KUKA KRL program: mixsort_main.src, mixsort_main.dat

--- mixsort_main.src ---
&ACCESS RVP
&REL 20
&COMMENT MixSort Main
&PARAM EDITMASK = *
&PARAM DISKPATH = KRC:\R1\Program\MixSortMain
DEF  mixsort_main ( )
;***********************************************************
;
; Copyright 2018 - 2025 speedbot All Rights reserved.
;
; File Name: mixsort_main.DAT
;
; Description:
;   Language             ==   Krl for KUKA ROBOT
;   Date                 ==   2022 - 06 - 27
;   Modification Data    ==   2025 - 02 - 10
;
; Author: speedbot
;
; Version: 1.1
;***********************************************************
;FOLD INI;%{PE}
    ;FOLD BASISTECH INI
        GLOBAL INTERRUPT DECL 3 WHEN $STOPMESS==TRUE DO IR_STOPM ( )
        INTERRUPT ON 3
        BAS (#INITMOV,0 )
    ;ENDFOLD (BASISTECH INI)
    ;FOLD USER INI
        ;Make your modifications here

    ;ENDFOLD (USER INI)
;ENDFOLD (INI)
;FOLD Basic.Override IN Override: 30  ;%{PE}
override_(30)
;ENDFOLD
;FOLD PLC.Pounce ;%{PE}
pounce_()
;ENDFOLD
mixsort_config()
;FOLD MixSort.MixSortSr ;%{PE}
mixsort_sr_inte()
;ENDFOLD
;FOLD MixSort.GetTask ;%{PE}
mixsort_get_task()
;ENDFOLD
LOOP
    continue
    wait for ToRobotFlg
    ToRobotFlg = false

    switch ToRobotAck
    case #TO_TP_NEXT
        mixsort_waitpos()
    case #TO_TP_PICT
        mixsort_picture()
    case #TO_TP_PK
        switch (GlobalTaskId)
        case 2
            mixsort_pick01()
        case 3
            mixsort_pick02()
        case 4
            mixsort_pick03()
        case 101
            mixsort_pick04()
        case 102
            mixsort_pick05()
        default
            log_error_("Unkonwn GlobalTaskId!")
        endswitch
        if (GlobalTaskId == 2) and (NOT $flag[F_PICKING]) THEN
            WAIT SEC 1
            mixsort_get_task()
        ELSE
            $flag[F_PICKING] = TRUE
            mixsort_place_select()
        ENDIF
    case #TO_TP_HOME
        exit
    endswitch
ENDLOOP
;FOLD PLC.MoveToHome ;%{PE}
move_to_home_()
;ENDFOLD
END

--- mixsort_main.dat ---
&ACCESS RVP
&REL 20
&COMMENT MixSort Main
&PARAM EDITMASK = *
&PARAM DISKPATH = KRC:\R1\Program\MixSortMain
DEFDAT  MIXSORT_MAIN
;***********************************************************
;
; Copyright 2018 - 2025 speedbot All Rights reserved.
;
; File Name: mixsort_main.DAT
;
; Description:
;   Language             ==   Krl for KUKA ROBOT
;   Date                 ==   2022 - 06 - 27
;   Modification Data    ==   2025 - 02 - 10
;
; Author: speedbot
;
; Version: 1.1
;***********************************************************
;FOLD EXTERNAL DECLARATIONS;%{PE}%MKUKATPBASIS,%CEXT,%VCOMMON,%P
;FOLD BASISTECH EXT;%{PE}%MKUKATPBASIS,%CEXT,%VEXT,%P
EXT  BAS (BAS_COMMAND  :IN,REAL  :IN )
EXT  mixsort_pick01 ( )
EXT  mixsort_pick02 ( )
EXT  mixsort_pick03 ( )
EXT  mixsort_pick04 ( )
EXT  mixsort_pick05 ( )
EXT  mixsort_place01 ( )
EXT  mixsort_place02 ( )
EXT  mixsort_place03 ( )
EXT  mixsort_place04 ( )
EXT  mixsort_place05 ( )
EXT  mixsort_place06 ( )
EXT  mixsort_place07 ( )
EXT  mixsort_place08 ( )
EXT  mixsort_drop01 ( )
EXT  mixsort_drop02 ( )
EXT  mixsort_drop03 ( )
EXT  mixsort_drop04 ( )
EXT  mixsort_picture ( )
EXT  mixsort_waitpos ( )

DECL INT SUCCESS
;ENDFOLD (BASISTECH EXT)
;FOLD USER EXT;%{E}%MKUKATPUSER,%CEXT,%VEXT,%P
;Make your modifications here

;ENDFOLD (USER EXT)
;ENDFOLD (EXTERNAL DECLARATIONS)

DECL part_data_t CopyPartData

DECL MODULEPARAM_T LAST_TP_PARAMS={PARAMS[] "BASIC.OVERRIDESPEED=30      "}
ENDDAT
